Omron CX-Programmer project NewProject (CX-Programmer 9.51)

# PLC my_first_project: CP1L L
; MyFirstProject

## Global symbols (name address type ; comment)
T0001 BOOL  ; Timer number

## Program NewProgram1 (cyclic task 0)
Local symbols
button_1 0.00 BOOL
out_3 100.02 BOOL

### Section Section1

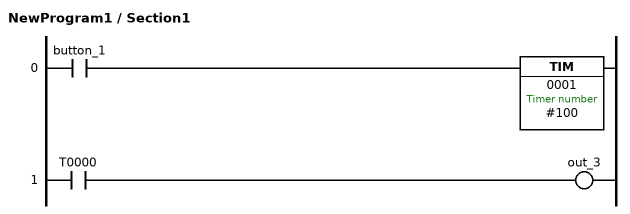
; rung 0
LD button_1
TIM 0001 #100  ; Timer number
; rung 1
LD T0000
OUT out_3

### Section END
; rung 0
END(001)